{attribute addProperty BoxType "EJ5002-0000-0017"}
{attribute addProperty Id "SSI_Inputs_ChannelAT %I*ARRAY[0..1] OF SSI_Inputs_Channel_32C7114D96120WcStateAT %I*WcState_F855686C1620InfoDataAT %I*InfoData_BC63D37F80100"}
{attribute addProperty CRC "3272543769"}
{attribute addProperty SizeInBites "192"}
{attribute addProperty SizeInBytes "24"}
TYPE EJ5002_D767A133 :
STRUCT
	{attribute addProperty Name "SSI_Inputs_Channel"}
	SSI_Inputs_Channel : ARRAY[0..1] OF SSI_Inputs_Channel_32C7114D;
	{attribute addProperty Name "WcState"}
	WcState : WcState_F855686C;
	{attribute addProperty Name "InfoData"}
	InfoData : InfoData_BC63D37F;
END_STRUCT
END_TYPE

(* stored: Version 1.2.0.0, ProductVersion 3.1.4024.9
   DUT EJ5002_D767A133: Id {1df13834-59fe-4b05-abca-74ef6e2d57e0} *)
